// TIA Portal V15.1 export
// export: Created 2024-05-17T05:38:29.0620807Z, ExportSetting WithDefaults, DisplayName Totally Integrated Automation Portal, DisplayVersion V15.1 Update 5, DisplayName TIA Portal Openness, DisplayVersion V15.1 Update 5, DisplayName SINAMICS Startdrive Advanced, DisplayVersion V15.1, DisplayName G130, G150, S120, S150, SINAMICS MV, S210, DisplayVersion V15.1, DisplayName G110M, G120, G120C, G120D, G120P, DisplayVersion V15.1, DisplayName STEP 7 Professional, DisplayVersion V15.1 Update 5, DisplayName STEP 7 Safety, DisplayVersion V15.1, DisplayName WinCC Professional, DisplayVersion V15.1 Update 5, DisplayName SIMATIC Visualization Architect, DisplayVersion V15.1
FUNCTION_BLOCK "L5Alarm"   // FB1405, FBD
TITLE = L5Alarm
{ S7_Optimized_Access := 'FALSE' }
AUTHOR : VCC
FAMILY : AlarmHnd
NAME : 5Alarm
VERSION : 1.0
// ================================================================================
// This module is used everywhere 5 alarms has to be generated when one (security) 
// corresponding input becomes True.
// All alarms can be True only when the corresponding input Enable Alarm is also 
// True.
// When the conditions to generate the alarm is disappear, a boolean (one per 
// alarm) available to inform the upper level that the corresponding alarm can be 
// reset.
// All alarms are reset by means of the AlarmResetPB signal.
// ================================================================================
// stored: AutoNumber false, IsIECCheckEnabled false, SetENOAutomatically False, UDAEnableTagReadback false
   VAR_INPUT
      I_Input1 { ExternalAccessible := 'False'; ExternalVisible := 'False'; ExternalWritable := 'False'} : Bool;   // Input alarm 1
      I_AlarmClass1 { ExternalAccessible := 'False'; ExternalVisible := 'False'; ExternalWritable := 'False'} : Char;   // Alarm class -> A - B - C - D or E
      I_EnableAlarm1 { ExternalAccessible := 'False'; ExternalVisible := 'False'; ExternalWritable := 'False'} : Bool := TRUE;   // Enable alarm 1 from upper level
      I_Invisible1 { ExternalAccessible := 'False'; ExternalVisible := 'False'; ExternalWritable := 'False'} : Bool;   // Invisible 1
      I_Input2 { ExternalAccessible := 'False'; ExternalVisible := 'False'; ExternalWritable := 'False'} : Bool;   // Input alarm 2
      I_AlarmClass2 { ExternalAccessible := 'False'; ExternalVisible := 'False'; ExternalWritable := 'False'} : Char;   // Alarm class -> A - B - C - D or E
      I_EnableAlarm2 { ExternalAccessible := 'False'; ExternalVisible := 'False'; ExternalWritable := 'False'} : Bool := TRUE;   // Enable alarm 2 from upper level
      I_Invisible2 { ExternalAccessible := 'False'; ExternalVisible := 'False'; ExternalWritable := 'False'} : Bool;   // Invisible 2
      I_Input3 { ExternalAccessible := 'False'; ExternalVisible := 'False'; ExternalWritable := 'False'} : Bool;   // Input alarm 3
      I_AlarmClass3 { ExternalAccessible := 'False'; ExternalVisible := 'False'; ExternalWritable := 'False'} : Char;   // Alarm class -> A - B - C - D or E
      I_EnableAlarm3 { ExternalAccessible := 'False'; ExternalVisible := 'False'; ExternalWritable := 'False'} : Bool := TRUE;   // Enable alarm 3 from upper level
      I_Invisible3 { ExternalAccessible := 'False'; ExternalVisible := 'False'; ExternalWritable := 'False'} : Bool;   // Invisible 3
      I_Input4 { ExternalAccessible := 'False'; ExternalVisible := 'False'; ExternalWritable := 'False'} : Bool;   // Input alarm 4
      I_AlarmClass4 { ExternalAccessible := 'False'; ExternalVisible := 'False'; ExternalWritable := 'False'} : Char;   // Alarm class -> A - B - C - D or E
      I_EnableAlarm4 { ExternalAccessible := 'False'; ExternalVisible := 'False'; ExternalWritable := 'False'} : Bool := TRUE;   // Enable alarm 4 from upper level
      I_Invisible4 { ExternalAccessible := 'False'; ExternalVisible := 'False'; ExternalWritable := 'False'} : Bool;   // Invisible 4
      I_Input5 { ExternalAccessible := 'False'; ExternalVisible := 'False'; ExternalWritable := 'False'} : Bool;   // Input alarm 5
      I_AlarmClass5 { ExternalAccessible := 'False'; ExternalVisible := 'False'; ExternalWritable := 'False'} : Char;   // Alarm class -> A - B - C - D or E
      I_EnableAlarm5 { ExternalAccessible := 'False'; ExternalVisible := 'False'; ExternalWritable := 'False'} : Bool := TRUE;   // Enable alarm 5 from upper level
      I_Invisible5 { ExternalAccessible := 'False'; ExternalVisible := 'False'; ExternalWritable := 'False'} : Bool;   // Invisible
      I_AlarmResetPB { ExternalAccessible := 'False'; ExternalVisible := 'False'; ExternalWritable := 'False'} : Bool;   // Alarm reset pushbutton is activated
   END_VAR
   VAR_OUTPUT
      O_Alarm1 { ExternalAccessible := 'False'; ExternalVisible := 'False'; ExternalWritable := 'False'} : Bool;   // Alarm 1
      O_Alarm2 { ExternalAccessible := 'False'; ExternalVisible := 'False'; ExternalWritable := 'False'} : Bool;   // Alarm 2
      O_Alarm3 { ExternalAccessible := 'False'; ExternalVisible := 'False'; ExternalWritable := 'False'} : Bool;   // Alarm 3
      O_Alarm4 { ExternalAccessible := 'False'; ExternalVisible := 'False'; ExternalWritable := 'False'} : Bool;   // Alarm 4
      O_Alarm5 { ExternalAccessible := 'False'; ExternalVisible := 'False'; ExternalWritable := 'False'} : Bool;   // Alarm 5
      O_AlarmABCondition { ExternalAccessible := 'False'; ExternalVisible := 'False'; ExternalWritable := 'False'} : Bool;   // Alarm AB condition
      H_IAnim1 { ExternalAccessible := 'False'; ExternalVisible := 'False'; ExternalWritable := 'False'} : Word;   // Icon Animation 1
      H_IAnim2 { ExternalAccessible := 'False'; ExternalVisible := 'False'; ExternalWritable := 'False'} : Word;   // Icon Animation 2
      H_IAnim3 { ExternalAccessible := 'False'; ExternalVisible := 'False'; ExternalWritable := 'False'} : Word;   // Icon Animation 3
      H_IAnim4 { ExternalAccessible := 'False'; ExternalVisible := 'False'; ExternalWritable := 'False'} : Word;   // Icon Animation 4
      H_IAnim5 { ExternalAccessible := 'False'; ExternalVisible := 'False'; ExternalWritable := 'False'} : Word;   // Icon Animation 5
   END_VAR
   VAR DB_SPECIFIC
      H_Out : Struct   // HMI
         Anim1 : Word;   // HMI Animation of the object
         Anim2 : Word;   // HMI Animation of the object
         Anim3 : Word;   // HMI Animation of the object
         Anim4 : Word;   // HMI Animation of the object
         Anim5 : Word;   // HMI Animation of the object
         DBnr : Int;   // HMI Animation DB number
      END_STRUCT;
      Alarm1 { ExternalAccessible := 'False'; ExternalVisible := 'False'; ExternalWritable := 'False'} : Bool;   // Alarm 1
      AlarmClass1_A { ExternalAccessible := 'False'; ExternalVisible := 'False'; ExternalWritable := 'False'} : Bool;   // The alarm is from alarm class A
      AlarmClass1_B { ExternalAccessible := 'False'; ExternalVisible := 'False'; ExternalWritable := 'False'} : Bool;   // The alarm is from alarm class B
      AlarmClass1_C { ExternalAccessible := 'False'; ExternalVisible := 'False'; ExternalWritable := 'False'} : Bool;   // The alarm is from alarm class C
      AlarmClass1_D { ExternalAccessible := 'False'; ExternalVisible := 'False'; ExternalWritable := 'False'} : Bool;   // The alarm is from alarm class D
      AlarmClass1_E { ExternalAccessible := 'False'; ExternalVisible := 'False'; ExternalWritable := 'False'} : Bool;   // The alarm is from alarm class E
      Alarm1Cond { ExternalAccessible := 'False'; ExternalVisible := 'False'; ExternalWritable := 'False'} : Bool;   // Alarm 1 condition
      Alarm2 { ExternalAccessible := 'False'; ExternalVisible := 'False'; ExternalWritable := 'False'} : Bool;   // Alarm 2
      AlarmClass2_A { ExternalAccessible := 'False'; ExternalVisible := 'False'; ExternalWritable := 'False'} : Bool;   // The alarm is from alarm class A
      AlarmClass2_B { ExternalAccessible := 'False'; ExternalVisible := 'False'; ExternalWritable := 'False'} : Bool;   // The alarm is from alarm class B
      AlarmClass2_C { ExternalAccessible := 'False'; ExternalVisible := 'False'; ExternalWritable := 'False'} : Bool;   // The alarm is from alarm class C
      AlarmClass2_D { ExternalAccessible := 'False'; ExternalVisible := 'False'; ExternalWritable := 'False'} : Bool;   // The alarm is from alarm class D
      AlarmClass2_E { ExternalAccessible := 'False'; ExternalVisible := 'False'; ExternalWritable := 'False'} : Bool;   // The alarm is from alarm class E
      Alarm2Cond { ExternalAccessible := 'False'; ExternalVisible := 'False'; ExternalWritable := 'False'} : Bool;   // Alarm 2 condition
      Alarm3 { ExternalAccessible := 'False'; ExternalVisible := 'False'; ExternalWritable := 'False'} : Bool;   // Alarm 3
      AlarmClass3_A { ExternalAccessible := 'False'; ExternalVisible := 'False'; ExternalWritable := 'False'} : Bool;   // The alarm is from alarm class A
      AlarmClass3_B { ExternalAccessible := 'False'; ExternalVisible := 'False'; ExternalWritable := 'False'} : Bool;   // The alarm is from alarm class B
      AlarmClass3_C { ExternalAccessible := 'False'; ExternalVisible := 'False'; ExternalWritable := 'False'} : Bool;   // The alarm is from alarm class C
      AlarmClass3_D { ExternalAccessible := 'False'; ExternalVisible := 'False'; ExternalWritable := 'False'} : Bool;   // The alarm is from alarm class D
      AlarmClass3_E { ExternalAccessible := 'False'; ExternalVisible := 'False'; ExternalWritable := 'False'} : Bool;   // The alarm is from alarm class E
      Alarm3Cond { ExternalAccessible := 'False'; ExternalVisible := 'False'; ExternalWritable := 'False'} : Bool;   // Alarm 3 condition
      Alarm4 { ExternalAccessible := 'False'; ExternalVisible := 'False'; ExternalWritable := 'False'} : Bool;   // Alarm 4
      AlarmClass4_A { ExternalAccessible := 'False'; ExternalVisible := 'False'; ExternalWritable := 'False'} : Bool;   // The alarm is from alarm class A
      AlarmClass4_B { ExternalAccessible := 'False'; ExternalVisible := 'False'; ExternalWritable := 'False'} : Bool;   // The alarm is from alarm class B
      AlarmClass4_C { ExternalAccessible := 'False'; ExternalVisible := 'False'; ExternalWritable := 'False'} : Bool;   // The alarm is from alarm class C
      AlarmClass4_D { ExternalAccessible := 'False'; ExternalVisible := 'False'; ExternalWritable := 'False'} : Bool;   // The alarm is from alarm class D
      AlarmClass4_E { ExternalAccessible := 'False'; ExternalVisible := 'False'; ExternalWritable := 'False'} : Bool;   // The alarm is from alarm class E
      Alarm4Cond { ExternalAccessible := 'False'; ExternalVisible := 'False'; ExternalWritable := 'False'} : Bool;   // Alarm 4 condition
      Alarm5 { ExternalAccessible := 'False'; ExternalVisible := 'False'; ExternalWritable := 'False'} : Bool;   // Alarm 5
      AlarmClass5_A { ExternalAccessible := 'False'; ExternalVisible := 'False'; ExternalWritable := 'False'} : Bool;   // The alarm is from alarm class A
      AlarmClass5_B { ExternalAccessible := 'False'; ExternalVisible := 'False'; ExternalWritable := 'False'} : Bool;   // The alarm is from alarm class B
      AlarmClass5_C { ExternalAccessible := 'False'; ExternalVisible := 'False'; ExternalWritable := 'False'} : Bool;   // The alarm is from alarm class C
      AlarmClass5_D { ExternalAccessible := 'False'; ExternalVisible := 'False'; ExternalWritable := 'False'} : Bool;   // The alarm is from alarm class D
      AlarmClass5_E { ExternalAccessible := 'False'; ExternalVisible := 'False'; ExternalWritable := 'False'} : Bool;   // The alarm is from alarm class E
      Alarm5Cond { ExternalAccessible := 'False'; ExternalVisible := 'False'; ExternalWritable := 'False'} : Bool;   // Alarm 5 condition
      DBnr { ExternalAccessible := 'False'; ExternalVisible := 'False'; ExternalWritable := 'False'} : Int;   // HMI DB number
   END_VAR
BEGIN

NETWORK
TITLE = **** 1 - Inputs **** DB number
// DB number
      L     DINO;
      T     #DBnr;

NETWORK
TITLE = **** 1 - Inputs **** Alarm class 1
// Alarm class
// Alarm class = E
      L     #I_AlarmClass1;
      L     'E';
      ==I;
      =     #AlarmClass1_E;

// Alarm class = D
      L     #I_AlarmClass1;
      L     'D';
      ==I;
      =     #AlarmClass1_D;

// Alarm class = C
      L     #I_AlarmClass1;
      L     'C';
      ==I;
      =     #AlarmClass1_C;

// Alarm class = B
      L     #I_AlarmClass1;
      L     'B';
      ==I;
      =     #AlarmClass1_B;

// Alarm class = A
      AN    #AlarmClass1_B;
      AN    #AlarmClass1_C;
      AN    #AlarmClass1_D;
      AN    #AlarmClass1_E;
      =     #AlarmClass1_A;


NETWORK
TITLE = **** 1 - Inputs **** Alarm class 2
// Alarm class
// Alarm class = E
      L     #I_AlarmClass2;
      L     'E';
      ==I;
      =     #AlarmClass2_E;

// Alarm class = D
      L     #I_AlarmClass2;
      L     'D';
      ==I;
      =     #AlarmClass2_D;

// Alarm class = C
      L     #I_AlarmClass2;
      L     'C';
      ==I;
      =     #AlarmClass2_C;

// Alarm class = B
      L     #I_AlarmClass2;
      L     'B';
      ==I;
      =     #AlarmClass2_B;

// Alarm class = A
      AN    #AlarmClass2_B;
      AN    #AlarmClass2_C;
      AN    #AlarmClass2_D;
      AN    #AlarmClass2_E;
      =     #AlarmClass2_A;


NETWORK
TITLE = **** 1 - Inputs **** Alarm class 3
// Alarm class
// Alarm class = E
      L     #I_AlarmClass3;
      L     'E';
      ==I;
      =     #AlarmClass3_E;

// Alarm class = D
      L     #I_AlarmClass3;
      L     'D';
      ==I;
      =     #AlarmClass3_D;

// Alarm class = C
      L     #I_AlarmClass3;
      L     'C';
      ==I;
      =     #AlarmClass3_C;

// Alarm class = B
      L     #I_AlarmClass3;
      L     'B';
      ==I;
      =     #AlarmClass3_B;

// Alarm class = A
      AN    #AlarmClass3_B;
      AN    #AlarmClass3_C;
      AN    #AlarmClass3_D;
      AN    #AlarmClass3_E;
      =     #AlarmClass3_A;


NETWORK
TITLE = **** 1 - Inputs **** Alarm class 4
// Alarm class
// Alarm class = E
      L     #I_AlarmClass4;
      L     'E';
      ==I;
      =     #AlarmClass4_E;

// Alarm class = D
      L     #I_AlarmClass4;
      L     'D';
      ==I;
      =     #AlarmClass4_D;

// Alarm class = C
      L     #I_AlarmClass4;
      L     'C';
      ==I;
      =     #AlarmClass4_C;

// Alarm class = B
      L     #I_AlarmClass4;
      L     'B';
      ==I;
      =     #AlarmClass4_B;

// Alarm class = A
      AN    #AlarmClass4_B;
      AN    #AlarmClass4_C;
      AN    #AlarmClass4_D;
      AN    #AlarmClass4_E;
      =     #AlarmClass4_A;


NETWORK
TITLE = **** 1 - Inputs **** Alarm class 5
// Alarm class
// Alarm class = E
      L     #I_AlarmClass5;
      L     'E';
      ==I;
      =     #AlarmClass5_E;

// Alarm class = D
      L     #I_AlarmClass5;
      L     'D';
      ==I;
      =     #AlarmClass5_D;

// Alarm class = C
      L     #I_AlarmClass5;
      L     'C';
      ==I;
      =     #AlarmClass5_C;

// Alarm class = B
      L     #I_AlarmClass5;
      L     'B';
      ==I;
      =     #AlarmClass5_B;

// Alarm class = A
      AN    #AlarmClass5_B;
      AN    #AlarmClass5_C;
      AN    #AlarmClass5_D;
      AN    #AlarmClass5_E;
      =     #AlarmClass5_A;


REGION Network 7: **** 2.2 - Alarms - Alarms Generation **** Alarm Condition 1
   // Condition for Alarm 1
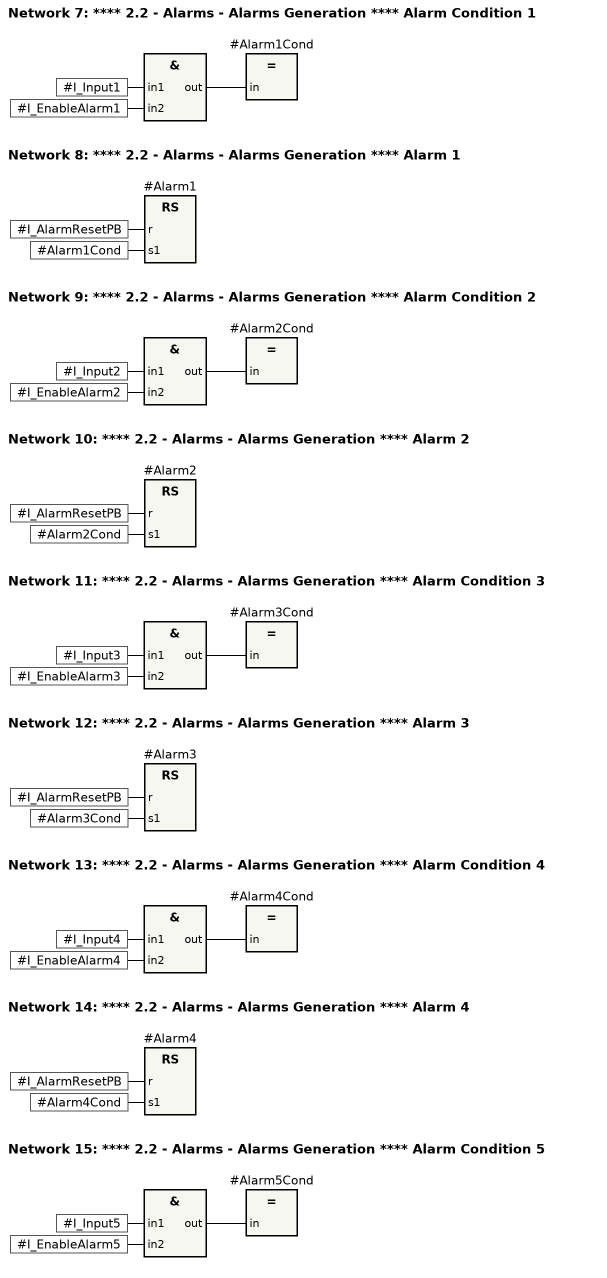
   #Alarm1Cond := #I_Input1 AND #I_EnableAlarm1;
END_REGION

REGION Network 8: **** 2.2 - Alarms - Alarms Generation **** Alarm 1
   // Creation of the Alarm 1
   IF #I_AlarmResetPB THEN
       #Alarm1 := FALSE;   // RS flip-flop
   END_IF;
   IF #Alarm1Cond THEN #Alarm1 := TRUE; END_IF;
END_REGION

REGION Network 9: **** 2.2 - Alarms - Alarms Generation **** Alarm Condition 2
   // Condition for Alarm 2
   #Alarm2Cond := #I_Input2 AND #I_EnableAlarm2;
END_REGION

REGION Network 10: **** 2.2 - Alarms - Alarms Generation **** Alarm 2
   // Creation of the Alarm 2
   IF #I_AlarmResetPB THEN
       #Alarm2 := FALSE;   // RS flip-flop
   END_IF;
   IF #Alarm2Cond THEN #Alarm2 := TRUE; END_IF;
END_REGION

REGION Network 11: **** 2.2 - Alarms - Alarms Generation **** Alarm Condition 3
   // Condition for Alarm 3
   #Alarm3Cond := #I_Input3 AND #I_EnableAlarm3;
END_REGION

REGION Network 12: **** 2.2 - Alarms - Alarms Generation **** Alarm 3
   // Creation of the Alarm 3
   IF #I_AlarmResetPB THEN
       #Alarm3 := FALSE;   // RS flip-flop
   END_IF;
   IF #Alarm3Cond THEN #Alarm3 := TRUE; END_IF;
END_REGION

REGION Network 13: **** 2.2 - Alarms - Alarms Generation **** Alarm Condition 4
   // Condition for Alarm 4
   #Alarm4Cond := #I_Input4 AND #I_EnableAlarm4;
END_REGION

REGION Network 14: **** 2.2 - Alarms - Alarms Generation **** Alarm 4
   // Creation of the Alarm 4
   IF #I_AlarmResetPB THEN
       #Alarm4 := FALSE;   // RS flip-flop
   END_IF;
   IF #Alarm4Cond THEN #Alarm4 := TRUE; END_IF;
END_REGION

REGION Network 15: **** 2.2 - Alarms - Alarms Generation **** Alarm Condition 5
   // Condition for Alarm 5
   #Alarm5Cond := #I_Input5 AND #I_EnableAlarm5;
END_REGION

REGION Network 16: **** 2.2 - Alarms - Alarms Generation **** Alarm 5
   // Creation of the Alarm 5
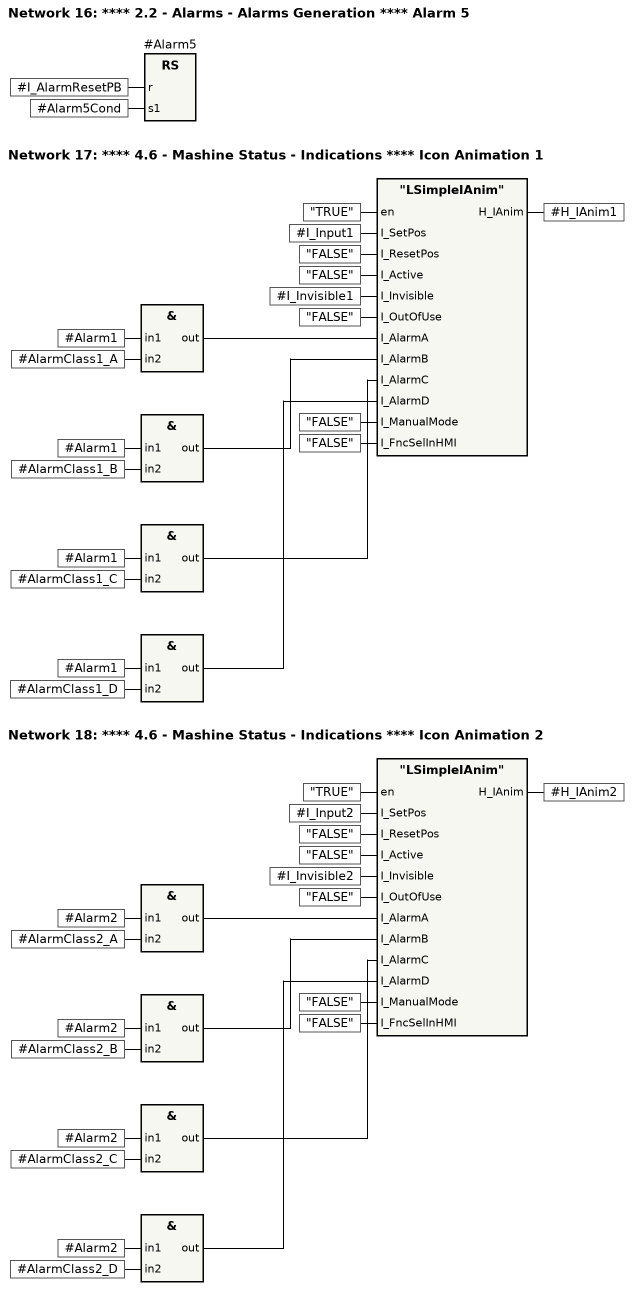
   IF #I_AlarmResetPB THEN
       #Alarm5 := FALSE;   // RS flip-flop
   END_IF;
   IF #Alarm5Cond THEN #Alarm5 := TRUE; END_IF;
END_REGION

REGION Network 17: **** 4.6 - Mashine Status - Indications **** Icon Animation 1
   // Icon Animation 1
   IF "TRUE" THEN
       "LSimpleIAnim"(I_SetPos := #I_Input1,
                      I_ResetPos := "FALSE",
                      I_Active := "FALSE",
                      I_Invisible := #I_Invisible1,
                      I_OutOfUse := "FALSE",
                      I_AlarmA := #Alarm1 AND #AlarmClass1_A,
                      I_AlarmB := #Alarm1 AND #AlarmClass1_B,
                      I_AlarmC := #Alarm1 AND #AlarmClass1_C,
                      I_AlarmD := #Alarm1 AND #AlarmClass1_D,
                      I_ManualMode := "FALSE",
                      I_FncSelInHMI := "FALSE",
                      H_IAnim => #H_IAnim1);
   END_IF;
END_REGION

REGION Network 18: **** 4.6 - Mashine Status - Indications **** Icon Animation 2
   // Icon Animation 2
   IF "TRUE" THEN
       "LSimpleIAnim"(I_SetPos := #I_Input2,
                      I_ResetPos := "FALSE",
                      I_Active := "FALSE",
                      I_Invisible := #I_Invisible2,
                      I_OutOfUse := "FALSE",
                      I_AlarmA := #Alarm2 AND #AlarmClass2_A,
                      I_AlarmB := #Alarm2 AND #AlarmClass2_B,
                      I_AlarmC := #Alarm2 AND #AlarmClass2_C,
                      I_AlarmD := #Alarm2 AND #AlarmClass2_D,
                      I_ManualMode := "FALSE",
                      I_FncSelInHMI := "FALSE",
                      H_IAnim => #H_IAnim2);
   END_IF;
END_REGION

REGION Network 19: **** 4.6 - Mashine Status - Indications **** Icon Animation 3
   // Icon Animation 3
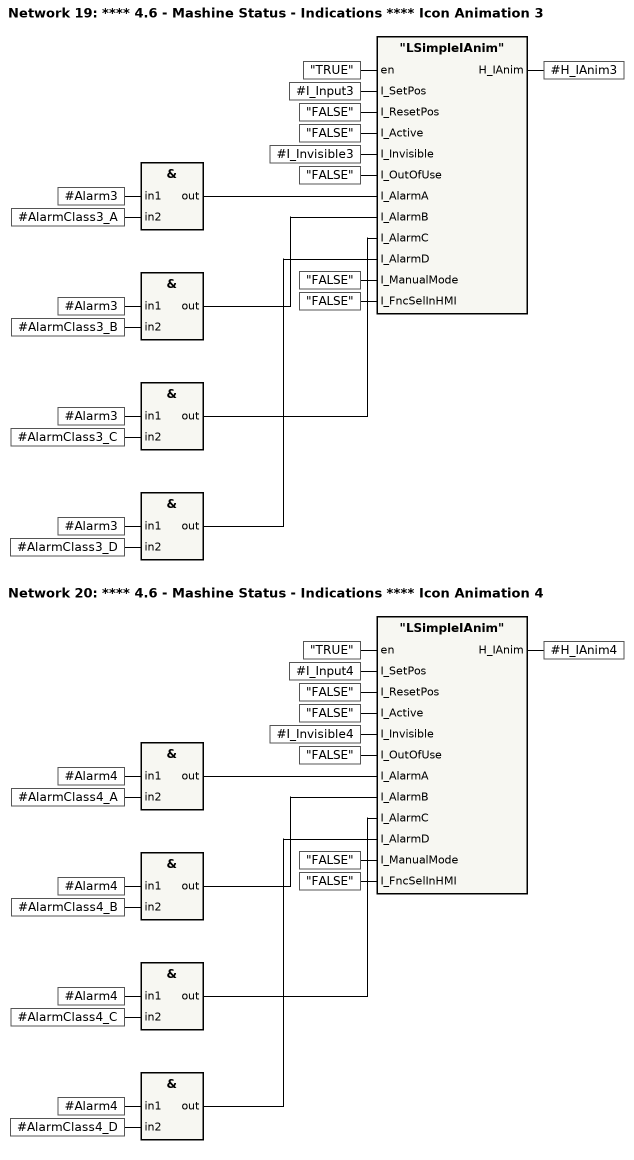
   IF "TRUE" THEN
       "LSimpleIAnim"(I_SetPos := #I_Input3,
                      I_ResetPos := "FALSE",
                      I_Active := "FALSE",
                      I_Invisible := #I_Invisible3,
                      I_OutOfUse := "FALSE",
                      I_AlarmA := #Alarm3 AND #AlarmClass3_A,
                      I_AlarmB := #Alarm3 AND #AlarmClass3_B,
                      I_AlarmC := #Alarm3 AND #AlarmClass3_C,
                      I_AlarmD := #Alarm3 AND #AlarmClass3_D,
                      I_ManualMode := "FALSE",
                      I_FncSelInHMI := "FALSE",
                      H_IAnim => #H_IAnim3);
   END_IF;
END_REGION

REGION Network 20: **** 4.6 - Mashine Status - Indications **** Icon Animation 4
   // Icon Animation 4
   IF "TRUE" THEN
       "LSimpleIAnim"(I_SetPos := #I_Input4,
                      I_ResetPos := "FALSE",
                      I_Active := "FALSE",
                      I_Invisible := #I_Invisible4,
                      I_OutOfUse := "FALSE",
                      I_AlarmA := #Alarm4 AND #AlarmClass4_A,
                      I_AlarmB := #Alarm4 AND #AlarmClass4_B,
                      I_AlarmC := #Alarm4 AND #AlarmClass4_C,
                      I_AlarmD := #Alarm4 AND #AlarmClass4_D,
                      I_ManualMode := "FALSE",
                      I_FncSelInHMI := "FALSE",
                      H_IAnim => #H_IAnim4);
   END_IF;
END_REGION

REGION Network 21: **** 4.6 - Mashine Status - Indications **** Icon Animation 5
   // Icon Animation 5
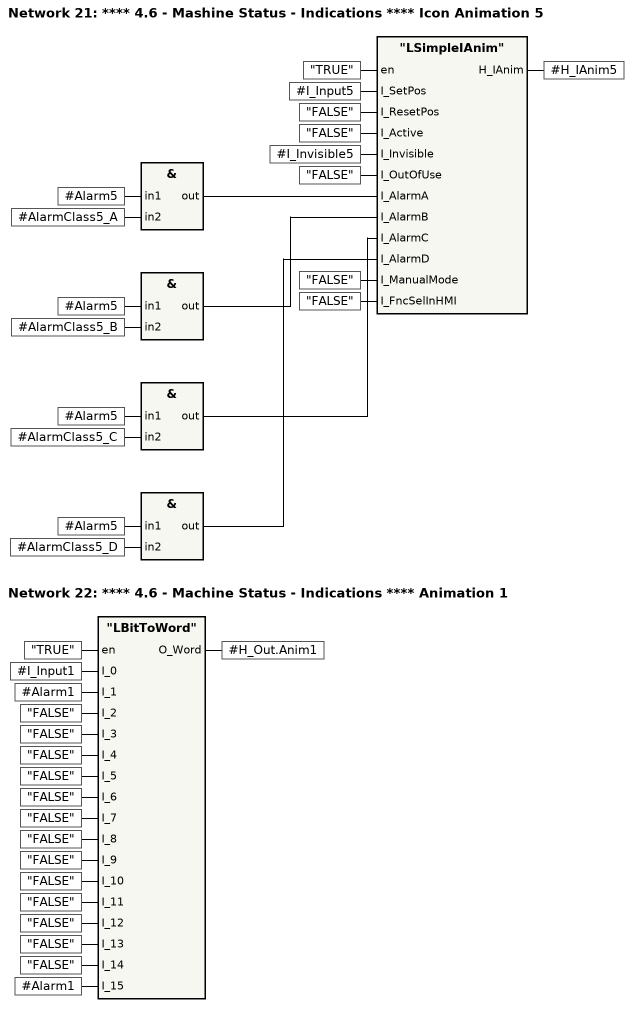
   IF "TRUE" THEN
       "LSimpleIAnim"(I_SetPos := #I_Input5,
                      I_ResetPos := "FALSE",
                      I_Active := "FALSE",
                      I_Invisible := #I_Invisible5,
                      I_OutOfUse := "FALSE",
                      I_AlarmA := #Alarm5 AND #AlarmClass5_A,
                      I_AlarmB := #Alarm5 AND #AlarmClass5_B,
                      I_AlarmC := #Alarm5 AND #AlarmClass5_C,
                      I_AlarmD := #Alarm5 AND #AlarmClass5_D,
                      I_ManualMode := "FALSE",
                      I_FncSelInHMI := "FALSE",
                      H_IAnim => #H_IAnim5);
   END_IF;
END_REGION

REGION Network 22: **** 4.6 - Machine Status - Indications **** Animation 1
   // Animation 1
   IF "TRUE" THEN
       "LBitToWord"(I_0 := #I_Input1,
                    I_1 := #Alarm1,
                    I_2 := "FALSE",
                    I_3 := "FALSE",
                    I_4 := "FALSE",
                    I_5 := "FALSE",
                    I_6 := "FALSE",
                    I_7 := "FALSE",
                    I_8 := "FALSE",
                    I_9 := "FALSE",
                    I_10 := "FALSE",
                    I_11 := "FALSE",
                    I_12 := "FALSE",
                    I_13 := "FALSE",
                    I_14 := "FALSE",
                    I_15 := #Alarm1,
                    O_Word => #H_Out.Anim1);
   END_IF;
END_REGION

REGION Network 23: **** 4.6 - Machine Status - Indications **** Animation 2
   // Animation 2
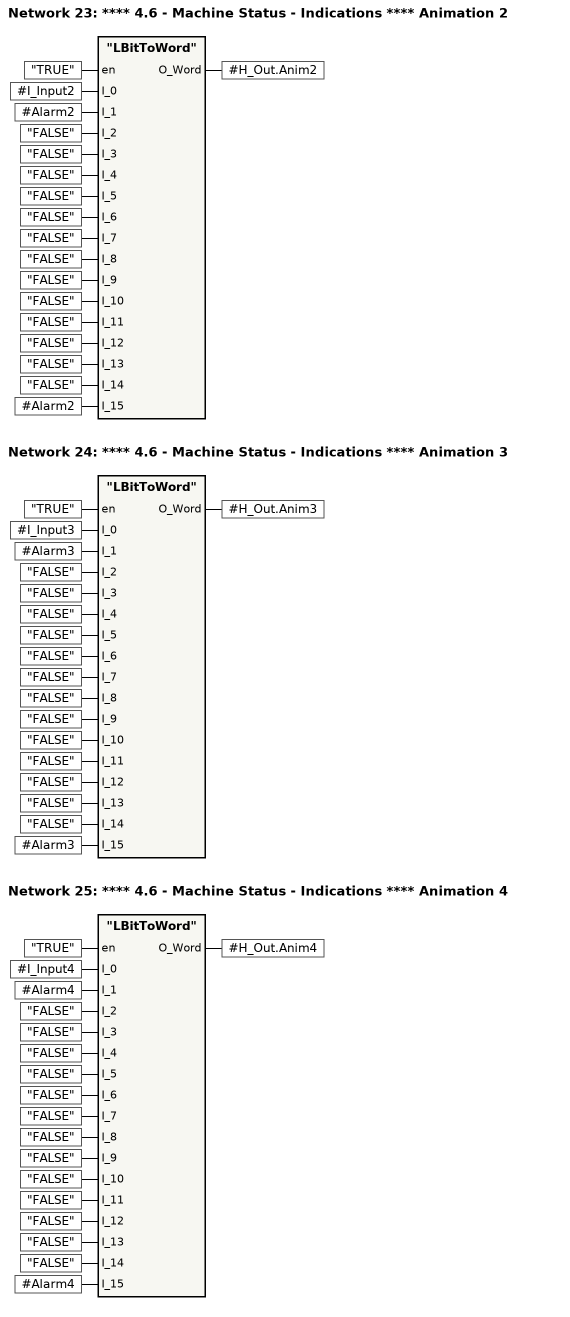
   IF "TRUE" THEN
       "LBitToWord"(I_0 := #I_Input2,
                    I_1 := #Alarm2,
                    I_2 := "FALSE",
                    I_3 := "FALSE",
                    I_4 := "FALSE",
                    I_5 := "FALSE",
                    I_6 := "FALSE",
                    I_7 := "FALSE",
                    I_8 := "FALSE",
                    I_9 := "FALSE",
                    I_10 := "FALSE",
                    I_11 := "FALSE",
                    I_12 := "FALSE",
                    I_13 := "FALSE",
                    I_14 := "FALSE",
                    I_15 := #Alarm2,
                    O_Word => #H_Out.Anim2);
   END_IF;
END_REGION

REGION Network 24: **** 4.6 - Machine Status - Indications **** Animation 3
   // Animation 3
   IF "TRUE" THEN
       "LBitToWord"(I_0 := #I_Input3,
                    I_1 := #Alarm3,
                    I_2 := "FALSE",
                    I_3 := "FALSE",
                    I_4 := "FALSE",
                    I_5 := "FALSE",
                    I_6 := "FALSE",
                    I_7 := "FALSE",
                    I_8 := "FALSE",
                    I_9 := "FALSE",
                    I_10 := "FALSE",
                    I_11 := "FALSE",
                    I_12 := "FALSE",
                    I_13 := "FALSE",
                    I_14 := "FALSE",
                    I_15 := #Alarm3,
                    O_Word => #H_Out.Anim3);
   END_IF;
END_REGION

REGION Network 25: **** 4.6 - Machine Status - Indications **** Animation 4
   // Animation 4
   IF "TRUE" THEN
       "LBitToWord"(I_0 := #I_Input4,
                    I_1 := #Alarm4,
                    I_2 := "FALSE",
                    I_3 := "FALSE",
                    I_4 := "FALSE",
                    I_5 := "FALSE",
                    I_6 := "FALSE",
                    I_7 := "FALSE",
                    I_8 := "FALSE",
                    I_9 := "FALSE",
                    I_10 := "FALSE",
                    I_11 := "FALSE",
                    I_12 := "FALSE",
                    I_13 := "FALSE",
                    I_14 := "FALSE",
                    I_15 := #Alarm4,
                    O_Word => #H_Out.Anim4);
   END_IF;
END_REGION

REGION Network 26: **** 4.6 - Machine Status - Indications **** Animation 5
   // Animation 5
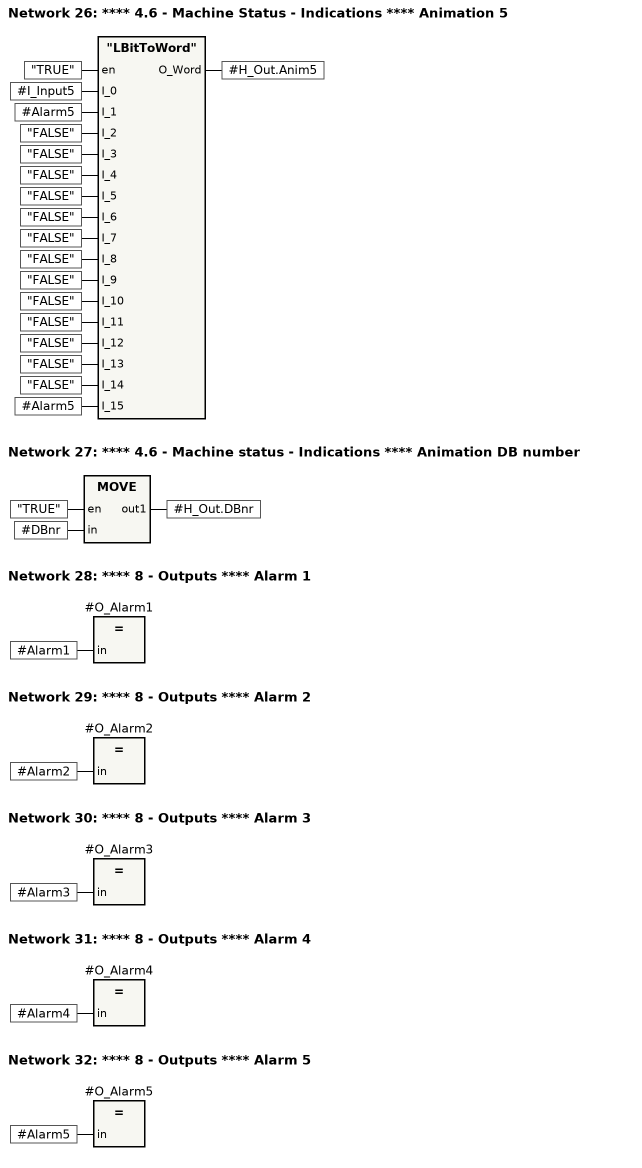
   IF "TRUE" THEN
       "LBitToWord"(I_0 := #I_Input5,
                    I_1 := #Alarm5,
                    I_2 := "FALSE",
                    I_3 := "FALSE",
                    I_4 := "FALSE",
                    I_5 := "FALSE",
                    I_6 := "FALSE",
                    I_7 := "FALSE",
                    I_8 := "FALSE",
                    I_9 := "FALSE",
                    I_10 := "FALSE",
                    I_11 := "FALSE",
                    I_12 := "FALSE",
                    I_13 := "FALSE",
                    I_14 := "FALSE",
                    I_15 := #Alarm5,
                    O_Word => #H_Out.Anim5);
   END_IF;
END_REGION

REGION Network 27: **** 4.6 - Machine status - Indications **** Animation DB number
   IF "TRUE" THEN #H_Out.DBnr := #DBnr; END_IF;
END_REGION

REGION Network 28: **** 8 - Outputs **** Alarm 1
   // Output of the Alarm 1
   #O_Alarm1 := #Alarm1;
END_REGION

REGION Network 29: **** 8 - Outputs **** Alarm 2
   // Output of the Alarm 2
   #O_Alarm2 := #Alarm2;
END_REGION

REGION Network 30: **** 8 - Outputs **** Alarm 3
   // Output of the Alarm 3
   #O_Alarm3 := #Alarm3;
END_REGION

REGION Network 31: **** 8 - Outputs **** Alarm 4
   // Output of the Alarm 4
   #O_Alarm4 := #Alarm4;
END_REGION

REGION Network 32: **** 8 - Outputs **** Alarm 5
   // Output of the Alarm 5
   #O_Alarm5 := #Alarm5;
END_REGION

REGION Network 33: **** 8 - Outputs **** Alarm AB Condition
   // Alarm AB condition
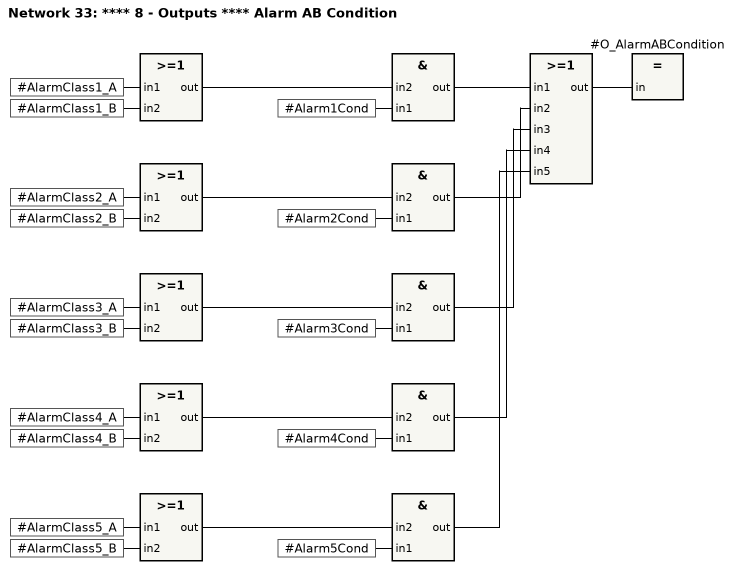
   #O_AlarmABCondition := ((#AlarmClass1_A OR #AlarmClass1_B) AND #Alarm1Cond) OR ((#AlarmClass2_A OR #AlarmClass2_B) AND #Alarm2Cond) OR ((#AlarmClass3_A OR #AlarmClass3_B) AND #Alarm3Cond) OR ((#AlarmClass4_A OR #AlarmClass4_B) AND #Alarm4Cond) OR ((#AlarmClass5_A OR #AlarmClass5_B) AND #Alarm5Cond);
END_REGION
END_FUNCTION_BLOCK
